Fanuc KAREL source: POST_SEMA.kl

PROGRAM T
%NOLOCKGROUP
VAR
 v0 : INTEGER
BEGIN
 POST_SEMA(v0)
END T
